# EPICS substitutions: scratchpad/tomostream_roi/iocBoot/iocEncoderStream_2BM/tomoStream.substitutions
file "$(TOP)/db/tomoStream.template"
{
pattern
{  P,      R, TOMO_SCAN, IMAGE_P, DARK_PVA, FLAT_PVA, RECON_PVA, THETA_PVA}
{2bmb:, EncoderStream:, 2bmb:TomoScanStream:, 2bmb:TomoScanStream:PvaPluginPVPrefix, 2bmb:TomoScanStream:StreamDarkFields, 2bmb:TomoScanStream:StreamFlatFields, 2bmb:EncoderStream:StreamRecon, 2bmb:TomoScanStream:StreamTheta}
}
